# EPICS autosave request: apps/xpsMotorApp/Db/motorsHallD.req
$(PREF)US1-2-BOT:m2:scan1.P1PA
$(PREF)US1-2-BOT:m2:scan1.P1SM
$(PREF)US1-2-BOT:m2:scan1.P1SP
$(PREF)US1-2-BOT:m2:scan1.P1EP
$(PREF)US1-2-BOT:m2:scan1.NPTS
$(PREF)US1-2-BOT:m2:saveData_scanNumber
$(PREF)US1-2-BOT:m2:saveData_fileSystem
$(PREF)US1-2-BOT:m2:saveData_subDir
$(PREF)US1-2-BOT:m2:saveData_baseName
$(PREF)US1-2-BOT:m2:scan1.PDLY
$(PREF)US1-2-BOT:m2:scan1.DDLY
